// TIA Portal V20 export
TYPE "UDT_Service_SupportedDigitalUnitSetting"
   STRUCT
      Unit { ExternalAccessible := 'False'; ExternalVisible := 'False'; ExternalWritable := 'False'} : Int := 1001;   // Supported Unit
      VMin { ExternalAccessible := 'False'; ExternalVisible := 'False'; ExternalWritable := 'False'} : DInt := 0;   // Value Low Limit
      VMax { ExternalAccessible := 'False'; ExternalVisible := 'False'; ExternalWritable := 'False'} : DInt := 100;   // Value High Limit
   END_STRUCT;
END_TYPE
